(* PLC project Unnamed, Unknown Unnamed 1 *)
(* stored: creationDateTime 2024-01-24T13:12:58, modificationDateTime 2024-01-29T11:01:01 *)

(* RawWaterPLC *)
PROGRAM RawWater
  VAR
    P101 AT %QX0.0 : BOOL;
    P102 AT %QX0.1 : BOOL;
    MV101 AT %QX0.2 : BOOL;
    FIT101 AT %MD0 : REAL;
    FIT201 AT %MD1 : REAL;
  END_VAR
  VAR CONSTANT
    ContainerMaxVolume AT %QW0 : INT := 1000;
  END_VAR
  VAR
    ContainerCurrentVolume AT %QW1 : INT;
  END_VAR

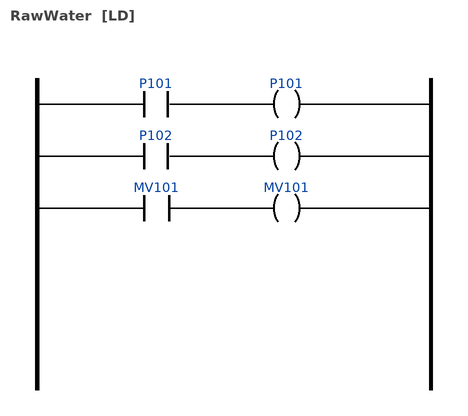
(* LD diagram, written out as Structured Text *)
P101 := P101;
P102 := P102;
MV101 := MV101;
END_PROGRAM

CONFIGURATION Config0
  RESOURCE Res0 ON PLC
    TASK task0(INTERVAL := T#20ms, PRIORITY := 0);
    PROGRAM instance0 WITH task0 : RawWater;
  END_RESOURCE
END_CONFIGURATION
